SUBAPPLICATION AR_TO_Q_Publish_OPC (* Physikalischer AR-Wert -> VT-Anzeige (Q_NumericValue_PHYSA) UND per OPC-UA publiziert (AR_PUBLISH_1), aus 1 gemeinsamer Quelle (AR_SPLIT_2). Fuer jeden Wert, der sowohl am VT angezeigt als auch lokal (Self-Subscribe) oder stationsuebergreifend weiterverwendet werden soll. *)
  (* Standard: 61499-2; Description: Copyright (c) 2026 Meisterschulen am Ostbahnhof This program and the accompanying materials are made available under the terms of the Eclipse Public License 2.0 which is available at https://www.eclipse.org/legal/epl-2.0/ SPDX-License-Identifier: EPL-2.0 *)
  (* Version 1.2, 2026-10-03, Franz Höpfinger, Meisterschulen am Ostbahnhof, Franz: RateLimit_Anzeige (AR_D_FF_TMIN) vor AR_SPLIT_2 verschoben (Absicht, nicht versehentlich) - drosselt jetzt BEIDE Zweige (VT-Anzeige UND AR_PUBLISH/Self-Subscribe-Konsumenten wie CTRL_PID_AR.AR_ACT) auf max. 1 Update/Tmin, statt nur die Anzeige. *)
  (* Version 1.1, 2026-10-03, Franz Höpfinger, Meisterschulen am Ostbahnhof, Franz: 'ich tendiere dazu weniger schnell die Anzeige zu aktualisieren und den Regler trotzdem schnell laufen zu lassen' (Kunde: traeges Verhalten bei eingeschalteter Aufnahme-Automatik, vermutlich VT-Bus-Last durch mehrere gleichzeitig schnell wechselnde Drehzahl-Anzeigen auf der Ernteseite) - 'AR_RATE_LIMIT haben wir schon, D_FF_TMIN': adapter::events::unidirectional::AR_D_FF_TMIN (Tmin=500ms) initial NUR auf dem VT-Anzeige-Zweig eingefuegt (v1.2 verschiebt ihn vor den Split, siehe dort). *)
  (* Version 1.0, 2026-09-12, Franz Höpfinger, Meisterschulen am Ostbahnhof, initial implementation - herausgeloest aus TECU_Speeds.SUB/TECU_RPTO.SUB (AR_SPLIT_2 + Q_NumericValue_PHYSA + AR_PUBLISH_1 kommt oft vor). *)
  PACKAGE MyLib::sys;
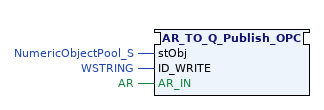
  VAR_INPUT
    stObj : logiBUS::utils::conversion::phys::NumericObjectPool_S; (* Object pool properties der VT-Zahlenvariable (u16ObjId, scale, offset, decimals) - z.B. FBs::const::DefaultPool_Numeric::NumberVariable_X_N *)
    ID_WRITE : WSTRING; (* Publish-Adresse (REAL, ACTION=PUBLISH), lokal oder stationsuebergreifend *)
  END_VAR
  SOCKETS
    AR_IN : adapter::types::unidirectional::AR; (* Physikalischer Wert (bereits skaliert) *)
  END_SOCKETS
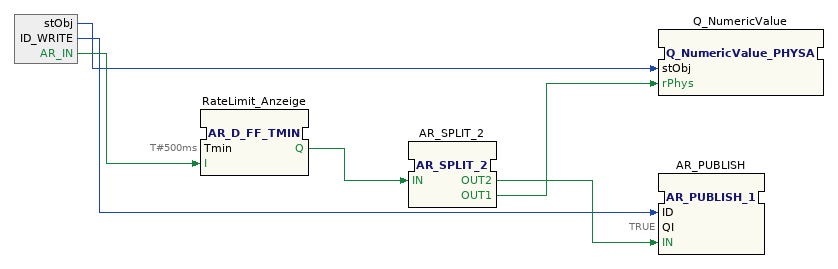
  FBS
    AR_SPLIT_2 : adapter::events::unidirectional::AR_SPLIT_2;
    RateLimit_Anzeige : adapter::events::unidirectional::AR_D_FF_TMIN(Tmin := T#500ms); (* Drosselt vor dem Split BEIDE Zweige (VT-Anzeige UND AR_PUBLISH/Self-Subscribe, z.B. CTRL_PID_AR.AR_ACT) auf max. 1 Update/500ms - Absicht (Franz). *)
    Q_NumericValue : isobus::UT::Q::Q_NumericValue_PHYSA;
    AR_PUBLISH : adapter::net::AR_PUBLISH_1(QI := TRUE);
  END_FBS
  DATA_CONNECTIONS
    stObj TO Q_NumericValue.stObj;
    ID_WRITE TO AR_PUBLISH.ID;
  END_CONNECTIONS
  ADAPTER_CONNECTIONS
    AR_IN TO RateLimit_Anzeige.I;
    AR_SPLIT_2.OUT2 TO AR_PUBLISH.IN;
    RateLimit_Anzeige.Q TO AR_SPLIT_2.IN;
    AR_SPLIT_2.OUT1 TO Q_NumericValue.rPhys;
  END_CONNECTIONS
END_SUBAPPLICATION
